FUNCTION_BLOCK EM_OutfeedA2 EXTENDS FB_Transport
FUNCTION_BLOCK EM_OutfeedA2 EXTENDS FB_Mechanische_Stop

VAR
	fb_mem : Str_FB_Transport;
END_VAR

END_FUNCTION_BLOCK

(* stored: Version 1.1.0.1, ProductVersion 3.1.4024.12
   POU EM_OutfeedA2: Id {785d883d-6312-4cfe-a0c5-3baf48e7776b}, SpecialFunc None *)
